(* Logix 5000 project; controller EuniceF_ICA18 vendor 1 type 14 code 150 rev 37.11; software revision 37.00 *)

TASK MainTask (continuous, watchdog 500 ms) : MainProgram

MODULES
   Local : vendor 1 type 14 code 150 (Compact 0, rev 37.11)
      Discrete_IO : Embedded (Compact 1, rev 3.1, Output RPI 20 ms)
      Analog_IO : Embedded (Compact 2, rev 1.1, Output RPI 80 ms)
      Counters : Embedded (Compact 3, rev 1.1, Output RPI 20 ms)
END_MODULES

VAR_GLOBAL   (* controller tags *)
   East_Green : BOOL;
   North_Red : BOOL;
   SEQ : DINT;
   Timer4s : TIMER := (PRE := 4000);
   Timer6s : TIMER := (PRE := 6000);
END_VAR

PROGRAM MainProgram   (* main routine MainRoutine *)

ROUTINE MainRoutine   (* ladder *)
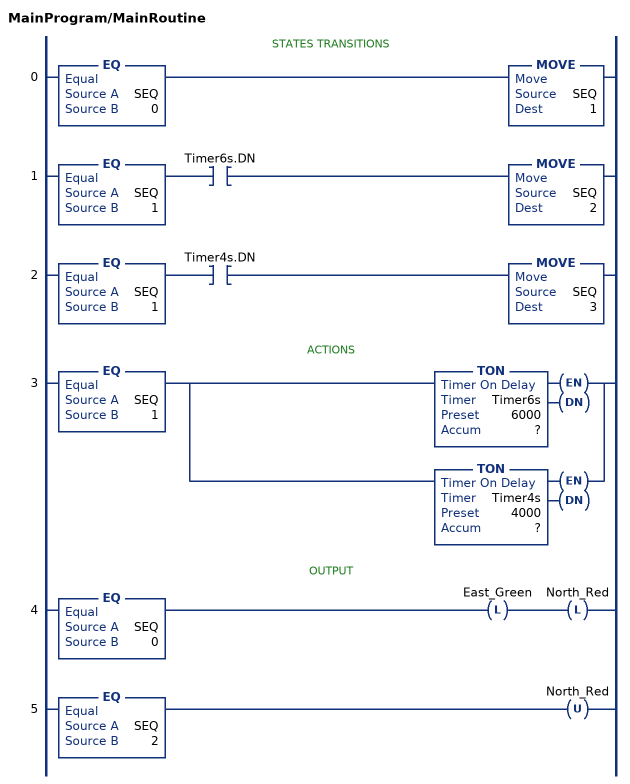
   // STATES TRANSITIONS
   0: EQ(SEQ,0)MOVE(SEQ,1);
   1: EQ(SEQ,1)XIC(Timer6s.DN)MOVE(SEQ,2);
   2: EQ(SEQ,1)XIC(Timer4s.DN)MOVE(SEQ,3);
   // ACTIONS
   3: EQ(SEQ,1)[TON(Timer6s,?,?) ,TON(Timer4s,?,?) ];
   // OUTPUT
   4: EQ(SEQ,0)OTL(East_Green)OTL(North_Red);
   5: EQ(SEQ,2)OTU(North_Red);
END_ROUTINE
END_PROGRAM
